TYPE ST_PlayerHelp :
STRUCT
	stBasicStrategy	: ST_BasicStrategy; //Basic strategy for playing common Black Jack 
END_STRUCT
END_TYPE

(* stored: Version 1.1.0.1, ProductVersion 3.1.4024.10
   DUT ST_PlayerHelp: Id {bff7f7e6-0b1a-4f4f-8d9a-56d2127cbcdc} *)
